KUKA KRL program: Mill_LeafHook3.src, Mill_LeafHook3.dat

--- Mill_LeafHook3.src ---
&ACCESS RVEO
&REL 5
&PARAM EDITMASK = *
&PARAM TEMPLATE = C:\KRC\Roboter\Template\vorgabe
&PARAM DISKPATH = KRC:\R1\Program\LeafProfiles
DEF Mill_LeafHook3( )
   ;FOLD DECL
      DECL ST_Dim3 stScrew[10],stPocket[3]
      DECL ST_Dim3 stScrewTemp,stPocketTemp
      DECL ST_Dim3 stHandle,stHandleTemp,stKey,stKeyTemp
      DECL INT iScrew,iPocket
   ;ENDFOLD
   ;FOLD INI

      ;stScrew[]
      FOR iScrew=1 TO iScrewSize STEP 1
         SetScrewData(iScrew,stScrewTemp)
         stScrew[iScrew] = stScrewTemp
      ENDFOR

      ;stPocket[]
      FOR iPocket=1 TO iPocketSize STEP 1
         SetPocketData(iPocket,stPocketTemp)
         stPocket[iPocket] = stPocketTemp
      ENDFOR

      ;stKey,stHandle
      SetHandleKeyData(stHandleTemp,stKeyTemp)
      stHandle = stHandleTemp
      stKey = stKeyTemp

   ;ENDFOLD

   TODO

   BAS(#INITMOV)

   ChangeStation(#AboveStations,#Idle)
   HALT

   ;Tool Cutter16
   ChangeStation(#ToolMagazine,#Idle)
   ToolMagazine(#Change,#SpindleHSD,#Cutter16)
   ChangeStation(#AboveStations,#Idle)
   HALT

   ;Handle, key milling
   ChangeStation(#MillHoriCenterHSD,#Idle)
   Spindle(#eRun,#SpindleHSD,17500)
   LeafMillHandle(stHandle)
   LeafMillKey(stKey)
   Spindle(#eStop)
   ChangeStation(#AboveStations,#Idle)
   HALT

   ;Pocket milling
   ChangeStation(#MillVertRightHSD,#Idle)
   Spindle(#eRun,#SpindleHSD,17500)
   MillLockPocket(stPocket[1],stAuxPocketDim,1)
   MillLockPocket(stPocket[2],stMainPocketDim,2)
   MillLockPocket(stPocket[3],stAuxPocketDim,1)
   Spindle(#eStop)
   ChangeStation(#AboveStations,#Idle)
   HALT

   ;Tool Drill3
   ChangeStation(#ToolMagazine,#Idle)
   ToolMagazine(#Change,#SpindleHSD,#Drill3)
   ChangeStation(#AboveStations,#Idle)
   HALT

   ;Screw drilling
   ChangeStation(#MillVertLeftHSD,#Idle)
   Spindle(#eRun,#SpindleHSD,6000)
   FOR iScrew=1 TO iScrewSize STEP 1
      DrillHole(#Drill3,stScrew[iScrew])
   ENDFOR
   Spindle(#eStop)
   ChangeStation(#AboveStations,#Idle,#MillVertRightHSD)

   ChangeStation(#HomePos,#Idle)

END

DEF SetScrewData(iScrew:IN,stScrewOut:OUT)
   ;FOLD DECL
      DECL INT iScrew,iScrewDAT
      DECL E_ProfilePlace eProfilePlace
      DECL E_ProfileType eProfileType
      DECL REAL rProfileLength
      DECL ST_Dim3 stScrewTemp,stScrewOut
   ;ENDFOLD (DECL)

   ;Take data from ProcessData structure
   eProfileType = gstProcessData.eProfileType
   eProfilePlace = gstProcessData.eProfilePlace
   rProfileLength = gstProcessData.rProfileLength

   ;DAT file screw number
   SWITCH eProfilePlace
      CASE #Left
         iScrewDAT = iScrewSize - (iScrew-1)
      CASE #Right
         iScrewDAT = iScrew
      DEFAULT
         HALT
   ENDSWITCH

   ;Take the right profile data
   SWITCH eProfileType
      CASE #Leaf75
         ;stScrewTemp = stScrewLeaf75[iScrewDAT]
      CASE #Leaf90
         stScrewTemp = stScrewLeaf90[iScrewDAT]
      DEFAULT
         HALT
   ENDSWITCH

   ;Initialization of screw data
   stScrewOut = stScrewTemp

   ;Correction of X coordinate
   SWITCH eProfilePlace
      CASE #Left
         stScrewOut.rX = grLongProfileRefX + stScrewTemp.rX
      CASE #Right
         stScrewOut.rX = grLongProfileRefX + rProfileLength - stScrewTemp.rX
      DEFAULT
         HALT
   ENDSWITCH

   ;Screw hole depth
   stScrewOut.rZ = rScrewHoleDepth

END

DEF SetPocketData(iPocket:IN,stPocketOut:OUT)
   ;FOLD DECL
      DECL INT iPocket,iPocketDAT
      DECL E_ProfilePlace eProfilePlace
      DECL E_ProfileType eProfileType
      DECL REAL rProfileLength
      DECL ST_Dim3 stPocketTemp,stPocketOut
   ;ENDFOLD (DECL)

   ;Take data from ProcessData structure
   eProfileType = gstProcessData.eProfileType
   eProfilePlace = gstProcessData.eProfilePlace
   rProfileLength = gstProcessData.rProfileLength

   ;DAT file pocket number
   SWITCH eProfilePlace
      CASE #Right
         iPocketDAT = iPocketSize - (iPocket-1)
      CASE #Left
         iPocketDAT = iPocket
      DEFAULT
         HALT
   ENDSWITCH

   ;Take the right profile data
   SWITCH eProfileType
      CASE #Frame75
         stPocketTemp = stPocketLeaf75[iPocketDAT]
      CASE #Frame90
         stPocketTemp = stPocketLeaf90[iPocketDAT]
      DEFAULT
         HALT
   ENDSWITCH

   ;Initialization of pocket data
   stPocketOut = stPocketTemp

   ;Correction of X coordiate
   SWITCH eProfilePlace
      CASE #Left
         stPocketOut.rX = grLongProfileRefX + stPocketTemp.rX
      CASE #Right
         stPocketOut.rX = grLongProfileRefX + rProfileLength - stPocketTemp.rX
      DEFAULT
         HALT
   ENDSWITCH

END

--- Mill_LeafHook3.dat ---
&ACCESS RVEO
&REL 5
&PARAM EDITMASK = *
&PARAM TEMPLATE = C:\KRC\Roboter\Template\vorgabe
&PARAM DISKPATH = KRC:\R1\Program\LeafProfiles
DEFDAT Mill_LeafHook3

   ;Amount of all screws
   DECL CONST INT iScrewSize = 10
   ;Depth of screw holes
   DECL CONST REAL rScrewHoleDepth = 6.0

   ;Screws Leaf75
   DECL ST_Dim3 stScrewLeaf75[10]
   stScrewLeaf75[1]  = {rX  163.0,rY 19.6,rZ 6.0}
   stScrewLeaf75[2]  = {rX  345.0,rY 19.6,rZ 6.0}
   stScrewLeaf75[3]  = {rX  518.0,rY 19.6,rZ 6.0}
   stScrewLeaf75[4]  = {rX  700.0,rY 19.6,rZ 6.0}
   stScrewLeaf75[5]  = {rX  855.0,rY 19.6,rZ 6.0}
   stScrewLeaf75[6]  = {rX 1130.0,rY 19.6,rZ 6.0}
   stScrewLeaf75[7]  = {rX 1298.0,rY 19.6,rZ 6.0}
   stScrewLeaf75[8]  = {rX 1480.0,rY 19.6,rZ 6.0}
   stScrewLeaf75[9]  = {rX 1653.0,rY 19.6,rZ 6.0}
   stScrewLeaf75[10] = {rX 1835.0,rY 19.6,rZ 6.0}

   ;Screws Leaf90
   DECL CONST ST_Dim3 stScrewLeaf90[10]
   stScrewLeaf90[1]  = {rX  168.0,rY 19.7,rZ 6.0}
   stScrewLeaf90[2]  = {rX  350.0,rY 19.7,rZ 6.0}
   stScrewLeaf90[3]  = {rX  523.0,rY 19.7,rZ 6.0}
   stScrewLeaf90[4]  = {rX  705.0,rY 19.7,rZ 6.0}
   stScrewLeaf90[5]  = {rX  860.0,rY 19.7,rZ 6.0}
   stScrewLeaf90[6]  = {rX 1135.0,rY 19.7,rZ 6.0}
   stScrewLeaf90[7]  = {rX 1303.0,rY 19.7,rZ 6.0}
   stScrewLeaf90[8]  = {rX 1485.0,rY 19.7,rZ 6.0}
   stScrewLeaf90[9]  = {rX 1658.0,rY 19.7,rZ 6.0}
   stScrewLeaf90[10] = {rX 1840.0,rY 19.7,rZ 6.0}

   ;Amount of all pockets
   DECL CONST INT iPocketSize = 3

   ;Pocket dimensions
   DECL CONST ST_Dim3 stAuxPocketDim  = {rX 130.0,rY 17.0}
   DECL CONST ST_Dim3 stMainPocketDim = {rX 200.0,rY 17.0}

   ;Pockets Leaf75
   DECL CONST ST_Dim3 stPocketLeaf75[3]
   stPocketLeaf75[1] = {rX  248.5,rY 19.6}
   stPocketLeaf75[2] = {rX  991.5,rY 19.6}
   stPocketLeaf75[3] = {rX 1738.5,rY 19.6}

   ;Pockets Leaf90
   DECL CONST ST_Dim3 stPocketLeaf90[3]
   stPocketLeaf90[1] = {rX  252.5,rY 19.7}
   stPocketLeaf90[2] = {rX  995.5,rY 19.7}
   stPocketLeaf90[3] = {rX 1742.5,rY 19.7}

ENDDAT
